FUNCTION_BLOCK ProductionAnalytics

VAR_IN_OUT
	DataArray 		: ARRAY[1..ARRAY_SIZE] OF REAL;   // Input array for analytics
END_VAR
VAR
	Idx       		: INT;                    		  // loop index 
END_VAR

VAR CONSTANT
	ARRAY_SIZE		: UINT := 10;
END_VAR

METHOD FindItem
VAR_INPUT
	SearchValue : REAL;             // The value to search for
    StartIndex  : UINT;            // Start index of the array to search in (1-based)
    EndIndex    : UINT;            // End index of the array to search in (1-based)
END_VAR

VAR_OUTPUT
    FoundIndex  : UINT;            // Index of the found value (1-based), 0 if not found
    Found       : BOOL;            // TRUE if the value is found, FALSE otherwise
    ValidInput  : BOOL;            // Indicates if the input parameters are valid
END_VAR

VAR
    MidIndex    : UINT;             // Midpoint index for binary search
    Low         : UINT;             // Lower boundary for search
    High        : UINT;             // Upper boundary for search
END_VAR
(* Find element using binary search algorithm *)

// Input validation
IF (StartIndex >= 1) AND (EndIndex <= ARRAY_SIZE) AND (StartIndex <= EndIndex) THEN
    ValidInput := TRUE;
ELSE
    ValidInput := FALSE;
    Found := FALSE;
    FoundIndex := 0;
    RETURN;
END_IF;

// Binary Search Algorithm
Low := StartIndex;
High := EndIndex;
Found := FALSE;       

WHILE (Low <= High) AND (NOT Found) DO
    // Calculate midpoint
    MidIndex := (Low + High) / 2;
    
    IF DataArray[MidIndex] = SearchValue THEN
        // Value found
        Found := TRUE;
        FoundIndex := MidIndex;
    ELSIF DataArray[MidIndex] < SearchValue THEN
        // Search in the right half
        Low := MidIndex + 1;
    ELSE
        // Search in the left half
        High := MidIndex - 1;
    END_IF;
END_WHILE;

// If not found, set FoundIndex to 0
IF NOT Found THEN
    FoundIndex := 0;  // Set to 0 to indicate not found
END_IF;
END_METHOD

METHOD GetMaxItem : REAL
VAR_INPUT
END_VAR

VAR
	ValidInput		: BOOL;
	SortedArray		: ARRAY[1..ARRAY_SIZE] OF REAL;
	IsSorted		: BOOL;
END_VAR
THIS^.Sort(SortedArray=>SortedArray, 
			IsSorted=>IsSorted, 
			ValidInput=>ValidInput);
			
If IsSorted then
	GetMaxItem := SortedArray[ARRAY_SIZE];
END_IF
END_METHOD

METHOD GetMean : REAL
VAR_INPUT
END_VAR

VAR
	Sum			: REAL;        // Sum of array elements 
	MeanTemp	: REAL;        // Temporary mean value for calculations
	Idx			: UINT;        // Loop counter 
END_VAR
(* Calculate the Mean *)

FOR Idx := 1 TO ARRAY_SIZE DO
	Sum := Sum + THIS^.DataArray[Idx];
END_FOR;


MeanTemp := Sum / TO_REAL(ARRAY_SIZE);
GetMean := MeanTemp;
END_METHOD

METHOD GetMinItem : REAL
VAR_INPUT
END_VAR

VAR
	ValidInput		: BOOL;
	SortedArray		: ARRAY[1..ARRAY_SIZE] OF REAL;
	IsSorted		: BOOL;
END_VAR
THIS^.Sort(SortedArray=>SortedArray, 
			IsSorted=>IsSorted, 
			ValidInput=>ValidInput);
			
If IsSorted then
	GetMinItem := SortedArray[1];
END_IF
END_METHOD

METHOD GetStdDev : REAL
VAR_INPUT
END_VAR

VAR
	MeanTemp		: REAL;		// Temporary mean value for calculations
	Deviation		: REAL;		// Deviation of each element from the mean
	SumOfSquares	: REAL;		// Sum of squared differences from the mean
	Idx				: UINT;     // Loop counter
	ArrayElement	: REAL;   	// Casted array element to REAL for precision
	MeanError		: BOOL;
END_VAR
(* Calculate the Standard Deviation *)

MeanTemp := THIS^.GetMean();

IF ARRAY_SIZE > 0 THEN
	FOR Idx := 1 TO ARRAY_SIZE DO
		ArrayElement := THIS^.DataArray[Idx];
		Deviation := ArrayElement - MeanTemp;						 
		SumOfSquares := SumOfSquares + (Deviation * Deviation); 
	END_FOR;

	GetStdDev := SQRT(SumOfSquares / TO_REAL(ARRAY_SIZE));
END_IF;
END_METHOD

METHOD GetTotal : REAL
VAR_INPUT
END_VAR

VAR
	Idx				: UINT;		// Loop counter
	ArrayElement	: REAL;		// Temporary array value	
	Total			: REAL;
END_VAR
FOR Idx := 1 TO ARRAY_SIZE DO
	ArrayElement := DataArray[Idx];
	Total := Total + ArrayElement;
END_FOR;

GetTotal := Total;
END_METHOD

METHOD Sort
VAR_INPUT
END_VAR

VAR_OUTPUT
    SortedArray   : ARRAY[1..ARRAY_SIZE] OF REAL;   // Output array with sorted elements
    IsSorted      : BOOL;                   // Indicates if the array is sorted
    ValidInput    : BOOL;                   // Indicates if the input parameters are valid
END_VAR

VAR
    Idx       	  : UINT;                   // Loop indices
    Parent, Child : UINT;                   // Indices for heap construction
    Temp          : REAL;                   // Temporary variable for swapping
END_VAR
(* Sort items using Heapsort algorithm*)

// --- Input Validation ---
IF (ARRAY_SIZE < 1) OR (ARRAY_SIZE > 100) THEN
    ValidInput := FALSE;
    IsSorted := FALSE;
    RETURN;
ELSE
    ValidInput := TRUE;
END_IF;

// --- Copy input array to output array ---
FOR Idx := 1 TO ARRAY_SIZE DO
    SortedArray[Idx] := THIS^.DataArray[Idx];
END_FOR;

// --- Heap Construction Phase ---
Idx := ARRAY_SIZE / 2;
WHILE Idx >= 1 DO
    Parent := Idx;
    WHILE 2 * Parent <= ARRAY_SIZE DO
        Child := 2 * Parent;
        
        // Select the larger child
        IF (Child < ARRAY_SIZE) AND 
			(SortedArray[Child] < SortedArray[Child + 1]) THEN
            Child := Child + 1;
        END_IF;
        
        // If parent is smaller than the largest child, swap them
        IF SortedArray[Parent] < SortedArray[Child] THEN
            Temp := SortedArray[Parent];
            SortedArray[Parent] := SortedArray[Child];
            SortedArray[Child] := Temp;
            
            // Move down the heap
            Parent := Child;
        ELSE
            EXIT;  // Break loop if the heap property is satisfied
        END_IF;
    END_WHILE;
    
    Idx := Idx - 1;  // Equivalent to DOWNTO without using DOWNTO
END_WHILE;

// --- Sorting Phase ---
FOR Idx := ARRAY_SIZE TO 2 BY -1 DO
    // Swap the first element (largest) with the last unsorted element
    Temp := SortedArray[1];
    SortedArray[1] := SortedArray[Idx];
    SortedArray[Idx] := Temp;
    
    // Restore the heap property for the reduced heap
    Parent := 1;
    WHILE 2 * Parent < Idx DO
        Child := 2 * Parent;
        
        // Select the larger child
        IF (Child < (Idx - 1)) AND (SortedArray[Child] < SortedArray[Child + 1]) THEN
            Child := Child + 1;
        END_IF;
        
        // If parent is smaller than the largest child, swap them
        IF SortedArray[Parent] < SortedArray[Child] THEN
            Temp := SortedArray[Parent];
            SortedArray[Parent] := SortedArray[Child];
            SortedArray[Child] := Temp;
            
            // Move down the heap
            Parent := Child;
        ELSE
            EXIT;  // Break loop if the heap property is satisfied
        END_IF;
    END_WHILE;
END_FOR;

// --- Set output signal to indicate sorting completion ---
IsSorted := TRUE;
END_METHOD

END_FUNCTION_BLOCK

(* stored: Version 1.1.0.1, ProductVersion 3.1.4024.15
   POU ProductionAnalytics: Id {b1bff168-853b-4299-a74a-90f79388f8db}, SpecialFunc None
   Method FindItem: Id {1411b85d-b0b6-457d-8e5c-27f03000bc3a}
   Method GetMaxItem: Id {5ad634df-d586-4f08-ad79-4f5375c07d8e}
   Method GetMean: Id {8c4778fa-c531-4d5f-b373-9543c70373dc}
   Method GetMinItem: Id {7456bce9-b437-4dcb-8a8b-0863e8851a7a}
   Method GetStdDev: Id {2445fe1d-db49-441a-a5cb-8b1dcd545cdc}
   Method GetTotal: Id {f486d8a5-2a48-42b6-980a-ea4f26827057}
   Method Sort: Id {20eba3b0-c28c-4818-8c39-d88bb54db329} *)
